PROGRAM P_BlinktaktTastleuchten
VAR
	//locByte0 : BYTE;
	blink:FB_MY_BLINK;
	blinkOld:BOOL := FALSE;
	b1HzOld:BOOL;
END_VAR

(* Netzwerk: 3 Blinktakt Tastleuchten - OK *)

//125 ms sind 8 Hz, mal sehen, ob ich die überhaupt brauche
blink(bEn := TRUE, udiTiOn_ms := 62, udiTiOff_ms := 63);

VAT.b1HzFlanke := FALSE;

IF blink.bQ <> blinkOld THEN
		
	VAT.byBlinkTakt := VAT.byBlinkTakt + 1;
	
	IO.outMldTasteStart :=	VAT.byBlinkTakt.0 AND // 8-Hz Blinktakt
							VAT.byBlinkTakt.1 AND // 4-Hz Blinktakt
							VAT.byBlinkTakt.2 AND // 2-Hz Blinktakt
							VAT.bEinzelSchritt
						 OR
							VAT.bSrStart AND
							NOT VAT.bSammelStoerung;
	
							
							
							
	IF b1HzOld <> VAT.byBlinkTakt.3 THEN
		VAT.b1HzFlanke := VAT.byBlinkTakt.3; //todo noch keine flanke
	END_IF	
	b1HzOld := VAT.byBlinkTakt.3;

	IF DB6.diStueck_Vorwahl > DB6.diStueck_Fertig THEN
		DB6.diStueck_Noch := DB6.diStueck_Vorwahl - DB6.diStueck_Fertig;
	END_IF						
END_IF

blinkOld := blink.bQ;

//IO.outResA1_2 := VAT.b1HzFlanke;


IF NOT VAT.b1HzFlanke THEN
	RETURN;
END_IF

//Verl. 5 Minuten für Betriebstunden-Zähler, todo Warum?

 


(*
	
		(*
			L 0
			T "MB 5" MB5 -- +F Blinktakt-Generator
		*)	
		VAT.M5 := 0;	
		(*	
			U "T 0" T0 -- Taktgeber
			SPB Takt -- Springe wenn VKE = 1
		*)	
		IF NOT GVL.T0.Q THEN
			(*
				L S5T#60MS
				SA "T 0" T0 -- Taktgeber
				CLR
				SA "T 0" T0 -- Taktgeber
			*)
			GVL.T0(IN := TRUE, PT := T#60MS);
			(*	
				L "MB 4" MB4 -- Blinktakt-Generator
				T LB 0
				INC 1
				T "MB 4" MB4 -- Blinktakt-Generator
				
				L LB 0
				INVI
				L "MB 4" MB4 -- Blinktakt-Generator
				UW
				
				T "MB 5" MB5 -- +F Blinktakt-Generator
			*)
			locByte0 := VAT.M4;
			VAT.M4 := VAT.M4 + 1;
			locByte0 := NOT locByte0;
			VAT.M5 := locByte0 AND VAT.M4;
			
			(*	
				U "M 4.0" M4.0 -- 8-Hz Blinktakt
				U "M 4.1" M4.1 -- 4-Hz Blinktakt
				U "M 4.2" M4.2 -- 2-Hz Blinktakt
				U "M0_3_Tipp" M0.3 -- Einzel-Schritt
				O "M0.6" M0.6 -- SR Start
				UN "M0.7" M0.7 -- Störung aufgetreten (gesammelt)
				= "A 0.0" A0.0 -- Tastleuchte Start
			*)	
			IO.outMldTasteStart :=	VAT.M4.0 AND // 8-Hz Blinktakt
									VAT.M4.1 AND // 4-Hz Blinktakt
									VAT.M4.2 AND // 2-Hz Blinktakt
									VAT.M0.3 OR  // Einzel-Schritt   
									VAT.M0.6 AND // SR Start
									NOT VAT.M0.7; // Störung aufgetreten (gesammelt)
			(*	
				L "DB6".d64Stueck_Vorwahl DB6.DBD64 -- Stückzahl-Vorwahl Stückz
				L "DB6".d68Stueck_Fertig DB6.DBD68 -- Fertig Stückz
				<D -- AKKU2 kleiner als AKKU1
				SPB Takt
				
				-D -- AKKU1 von AKKU2 subtrahieren
				T "DB6".d72Stueck_Noch DB6.DBD72 -- Noch Stückzahl
			*)
			IF DB6.d64Stueck_Vorwahl > DB6.d68Stueck_Fertig THEN
				DB6.d72Stueck_Noch := DB6.d64Stueck_Vorwahl - DB6.d68Stueck_Fertig;
			END_IF
		ELSE
			GVL.T0(IN := FALSE);	
		END_IF	//end if NOT GVL.T0.Q...
		
		(*	
		Takt: BLD 130
			U "M 5.3" M5.3 -- +F 1-Hz Blinktakt
			SPBN bz
		*)	
		IF NOT VAT.M5.3 THEN
			RETURN;
		END_IF
*)


		
(*
	U "T 34" T34 -- Verl. 5 Minuten für Betriebstunden-Zähler
	SPBN bz
*)
IF NOT GVL.tofBetrStdZaehl.Q THEN
	RETURN;
END_IF
	
(*	
	L "DB6".d160 DB6.DBD160 -- Betriebs-Sekunden
	+ L#1
	T "DB6".d160 DB6.DBD160 -- Betriebs-Sekunden
	L L#3600
	<D -- AKKU2 kleiner als AKKU1
	SPB bz
*)
	
DB6.runTime.seconds := DB6.runTime.seconds + 1;
IF DB6.runTime.seconds < 3600 THEN
	RETURN;
END_IF
	
(*	
	L 0
	T "DB6".d160 DB6.DBD160 -- Betriebs-Sekunden
*)	
DB6.runTime.seconds := 0;
(*	
	L "DB6".d164_Betriebs_St DB6.DBD164 -- Betriebs-Stunden
	+ L#1
	T "DB6".d164_Betriebs_St DB6.DBD164 -- Betriebs-Stunden
*)
DB6.runTime.hours := DB6.runTime.hours  + 1;
(*	
bz: BLD 130
*)

END_PROGRAM

(* stored: Version 1.1.0.1, ProductVersion 3.1.4024.3
   POU P_BlinktaktTastleuchten: Id {6c5c6349-eff9-41a1-a3a1-4d2d046f67d0}, SpecialFunc None *)
